INTERFACE ITcoCylinder EXTENDS __System.IQueryInterface

PROPERTY AtHome : bool
GET
END_GET
END_PROPERTY

PROPERTY AtWork : bool
GET
END_GET
END_PROPERTY

METHOD MoveToHome : TcoCore.ITcoTaskStatus
END_METHOD

METHOD MoveToWork :TcoCore.ITcoTaskStatus
END_METHOD

(*~
	<docu>
		<summary>
			Stops cyclinder movement.
		 	<remarks>			
				<note type="important">
					This method switched off the signals for the movement of the piston in both direction.
					However depending on the pnemumatics configuration the movement may contintue if designed in that way.
					THIS IS NOT A SAFETY FUCTION!
				</note>
			</remarks>	 		
		</summary>			
	</docu>	
~*)
METHOD Stop : TcoCore.ITcoTaskStatus
END_METHOD

END_INTERFACE

(* stored: Version 1.1.0.1
   Itf ITcoCylinder: Id {f5fb744e-8a3c-4ca5-afc7-036cd2bd31fb}
   Folder Actions: Id {1111bead-4c16-0549-0311-8f8313ecdb08}
   Folder States: Id {7060230d-ab76-0497-1872-fe660cbd877c}
   Property AtHome: Id {692c9f1a-d5e3-4f4a-9a9a-282429eb8537}
   Get Get: Id {e9381276-183c-4554-9e0d-6f5dae55cf75}
   Property AtWork: Id {659097f8-ff2d-44da-ad8a-231bc9f0b243}
   Get Get: Id {835540d8-d675-47f7-a931-ab492f87d3c7}
   Method MoveToHome: Id {b451c53c-b8b3-0c87-06bd-aa96c0705a24}
   Method MoveToWork: Id {d4c6ed9e-770f-0637-0124-63ecf1fb79b7}
   Method Stop: Id {e8983942-2e0e-0d6d-2470-ebd98bdb8f55} *)
